FUNCTION_BLOCK FbSetReset
VAR_INPUT
	xSet: BOOL;
	xReset: BOOL;
END_VAR
VAR_OUTPUT
	/// Memory 
	xQ: BOOL;
END_VAR

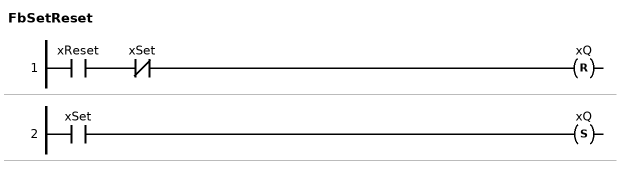
// NETWORK 1
xQ R= xReset AND NOT xSet;

// NETWORK 2
xQ S= xSet;

END_FUNCTION_BLOCK

(* stored: Version 1.1.0.1, ProductVersion 3.1.4024.12
   POU FbSetReset: Id {75dc1276-897f-491f-a31d-cea4348e1f71}, SpecialFunc None *)
